RoboDK station: Conveyor Simulation.rdk

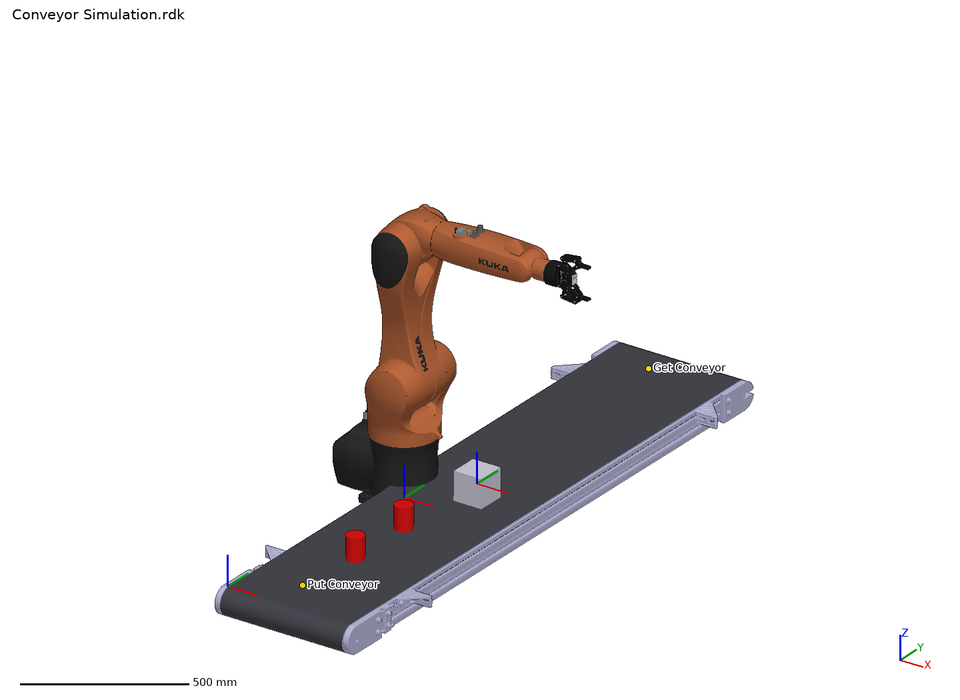
[picture v0: the station drawn from its stored meshes, robots at their saved joint values, targets as dots, program paths as lines]
Station Conveyor Simulation. Poses are relative to the parent item; angles as X-Y-Z fixed-axis rotations.
  - frame KUKA KR 10 R900 sixx Base at (-17.88, 1337.47, -86.35) mm
    - robot KUKA KR 10 R900 sixx: 6 axes, payload 10 kg, reach 901 mm, repeatability 0.03 mm, weight 52 kg
        modified DH rows (alpha deg, a mm, theta deg, d mm): 0, 0, 0, 400; -90, 25, 0, 0; 0, 455, -90, 0; -90, 35, 0, 420; 90, 0, 0, 0; -90, 0, 180, 80
        joint limits [-170, -190, -120, -185, -120, -350] to [170, 45, 156, 185, 120, 350]; home [0, -90, 90, 0, 0, 0]; saved at [0, -90, 90, 0, 0, 0]
      - tool Gripper RobotiQ 85 Opened, TCP at (0, 0, 130) mm, size 147.4 x 146.8 x 75 mm
  - frame ConveyorReference at (0, 403.83, 0) mm
    - target Get Conveyor (Cartesian target) at (200, 1882.78, 20) mm, rotated rx 90 ry 0 rz 0 deg; joints [0, 0, 0, 0, 0, 43.699]
    - target Put Conveyor (Cartesian target) at (200, 100, 20) mm, rotated rx 90 ry 0 rz -180 deg; joints [134.006, 22.86, -66.558, 43.699, -45.994, 0]
    - object Conveyor at (0, 300, -50) mm, size 597 x 2090.8 x 107.2 mm
      - Python program RunConveyor (listed below)
      - Python program WaitForPart (listed below)
      - Python program SimulateGripper (listed below)
    - object Part 1 at (200, 369.41, 40) mm, size 60 x 60 x 80 mm
    - object Part 2 at (200, 619.38, 40) mm, size 60 x 60 x 80 mm
  - frame Frame 3 at (262.28, 1312.72, 47.33) mm
    - object box at (0, 0, 0) mm, size 100 x 100 x 100 mm, geometry from box.sld

--- Python program RunConveyor ---
# Type help("robolink") or help("robodk") for more information
# Press F5 to run the script
# Note: you do not need to keep a copy of this file, your python script is saved with the station
from robolink import *    # API to communicate with RoboDK
from robodk import *      # basic matrix operations
RDK = Robolink()

# This script simulates a conveyor belt
CONVEYOR_NAME = 'Conveyor'
PICKABLE_OBJECTS_KEYWORD = 'Part'

# Speed of movement in MM/S with respect to the conveyor coordinates:
MOVE_SPEED_MMS = [0,5,0]
REFRESH_RATE = 0.005

# Define workspace of the conveyor to pick the objects:
CONV_SZ_X_MIN = 0
CONV_SZ_X_MAX = 440
CONV_SZ_Y_MIN = 0
CONV_SZ_Y_MAX = 2000
CONV_SZ_Z_MIN = -200
CONV_SZ_Z_MAX = +500

# Move objects that reached the end of the conveyor and were not picked:
FALLEN_OBJECTS = [0,0,-500]

# Get the conveyor item and reference for work space:
conv = RDK.Item(CONVEYOR_NAME)
conv_reference = conv.Parent()
poseconv = conv_reference.PoseAbs()

# One second in real life means 1 second of simulation. The simulation speed is taken from the station
SIMULATION_SPEED = 1

def is_inside_conveyor(pose):
    """Checks if a pose is inside the conveyor workspace"""
    pos = pose.Pos()
    if pos[0] > CONV_SZ_X_MIN and pos[0] < CONV_SZ_X_MAX and pos[1] > CONV_SZ_Y_MIN and pos[1] < CONV_SZ_Y_MAX and pos[2] > CONV_SZ_Z_MIN and pos[2] < CONV_SZ_Z_MAX:
        return True
    return False

def conveyor_move_object(pose, delta_time):
    """Moves the object pose through the conveyor depending on the time and speed"""
    delta_mm = mult3(MOVE_SPEED_MMS, delta_time)
    newpose = transl(delta_mm)*pose
    return newpose

# Get all objects (string list)
all_objects = RDK.ItemList(ITEM_TYPE_OBJECT, True)

# Convert object list into item pointers (faster)
# Also filter the list to take into account pickable objects only
objects = []
objects_name = []
objects_active = []
for i in range(len(all_objects)):
    if all_objects[i].count(PICKABLE_OBJECTS_KEYWORD) > 0:
        objects.append(RDK.Item(all_objects[i]))
        objects_name.append(all_objects[i])
        objects_active.append(False)

# The number of objects that can go in the conveyor
nobjects = len(objects)


# Infinite loop to simulate the conveyor behavior
current_time = 0
tic()
time_last = toc()
while True:
    # First: Look for objects that are not in the conveyor but are in the conveyor workspace
    for i in range(nobjects):
        obj_i = objects[i]

        # Skip if the object is already in the conveyor
        if objects_active[i]:
            continue

        # Check if the object has already been taken by a tool. If so, do not take it in the conveyor
        if obj_i.Parent().Type() == ITEM_TYPE_TOOL:
            continue

        # Check if the object is within the conveyor work area
        posei = obj_i.PoseAbs()
        poseirel = invH(poseconv)*posei
        if is_inside_conveyor(poseirel):
            # take the object
            obj_i.setParentStatic(conv)
            print('Adding object %s to the conveyor' % objects_name[i])
            objects_active[i] = True

    # Second step: Update the position of every object in the conveyor
    SIMULATION_SPEED = RDK.SimulationSpeed()
    time_current = toc()
    time_delta = time_current - time_last
    time_last = time_current
    current_time = current_time + time_delta*SIMULATION_SPEED

    # Make a list of objects with their matching positions to update
    obj_items = []
    obj_poses_abs = []
    for i in range(nobjects):
        obj_i = objects[i]

        # Check if the object has been picked from the conveyor
        if objects_active[i] and not obj_i.Parent().equals(conv):
            objects_active[i] = False
            print('Object %s was picked from the conveyor' % objects_name[i])
            continue

        # Skip update for objects that are not in the conveyor
        if not objects_active[i]:
            continue

        # Update the position of the object
        posei = invH(poseconv)*obj_i.PoseAbs()
        newposei = conveyor_move_object(posei, time_delta*SIMULATION_SPEED)
        if not is_inside_conveyor(newposei):
            print('Warning!! Object %s fell from the conveyor at %.1f seconds after simulation started' % (objects_name[i], current_time))
            #raise Exception('Object %s was not picked from the conveyor!' % objects_name[i])
            newposei = transl(FALLEN_OBJECTS)*newposei
            objects_active[i] = False

        #obj_i.setPose(newposei) # this will provoke a refresh (can be slow)
        obj_items.append(obj_i)
        obj_poses_abs.append(poseconv*newposei)

    # Update the object positions
    RDK.setPosesAbs(obj_items, obj_poses_abs)

    # Take a break...
    pause(REFRESH_RATE)

--- Python program WaitForPart ---
# Type help("robolink") or help("robodk") for more information
# Press F5 to run the script
# Note: you do not need to keep a copy of this file, your python script is saved with the station
from robolink import *    # API to communicate with RoboDK
from robodk import *      # basic matrix operations
RDK = Robolink()

# This script allows to simulate a laser sensor
# that detect the presence of a part in a plane,
# such as a part crossing a laser sensor in a
# conveyor belt

# The script finishes once a part has been detected
# so it works like a WAIT UNTIL function.

# Use a target from the station as a reference plane:
TARGET_NAME = 'Get Conveyor'
LASER_PLANE = [0,-1,0] # normal of the plane

# Activate within this tolerance
TOLERANCE_CHECK_MM = 10

# Look for parts with the keyword "Part"
PICKABLE_OBJECTS_KEYWORD = 'Part'

# Update status every 1 ms
RECHECK_PERIOD = 0.001

# Get the target and the detection plane
target = RDK.Item(TARGET_NAME)
targetpose = target.PoseAbs()
DETECT_PLANE_POINT = targetpose.Pos()
DETECT_PLANE_VECTOR = LASER_PLANE

# Define a function to detect a target
def part_detected(pos):
    """Check if a part is in the detection area (proximity of a point to a plane)"""
    pos_proj = proj_pt_2_plane(pos, DETECT_PLANE_POINT, DETECT_PLANE_VECTOR)
    distance2plane = norm(subs3(pos,pos_proj))
    if distance2plane < TOLERANCE_CHECK_MM:
        return True
    return False

# Get all object names
all_objects = RDK.ItemList(ITEM_TYPE_OBJECT, True)

# Get object items in a list (faster) and filter by keyword
check_objects = []
check_objects_names = []
for i in range(len(all_objects)):
    if all_objects[i].count(PICKABLE_OBJECTS_KEYWORD) > 0:
        check_objects_names.append(all_objects[i])
        check_objects.append(RDK.Item(all_objects[i]))

# Make sure that there are part that we are expecting
nCheck_objects = len(check_objects)
if nCheck_objects == 0:
    raise Exception('No parts to check for. The keyword is %s.' % PICKABLE_OBJECTS_KEYWORD)

# Loop forever until a part is detected by the sensor
part_available = False;
while not part_available:
    for i in range(nCheck_objects):
        if part_detected(check_objects[i].PoseAbs().Pos()):
            print('Part detected: %s' % check_objects_names[i])
            part_available = True
            break

    # Wait some time...
    pause(RECHECK_PERIOD)

print('Procedure finished')

--- Python program SimulateGripper ---
# Type help("robolink") or help("robodk") for more information
# Press F5 to run the script
# Note: you do not need to keep a copy of this file, your python script is saved with the station
from robolink import *    # API to communicate with RoboDK
from robodk import *      # basic matrix operations
RDK = Robolink()

# This file allows simulating the opening and closing of grippers.
# Two models of the gripper per robot are required: one opened and one closed.
# The opened model of the gripper should have the keyword "Opened"
# The closed model of the gripper should have the keyword "Closed"
# Simply place this file in the station and leave it running to
# make it work

OPENED_KEYWORD = 'Opened'
CLOSED_KEYWORD = 'Closed'
UPDATE_FREQUENCY = 0.01

# Loop forever
print('Starting infinite loop to simulate open/close of tools')
while True:
    # First step: get a list of tool pairs (open, closed) per robot
    Tool_Pairs = []
    # get all the robot names (strings)
    all_robots = RDK.ItemList(ITEM_TYPE_ROBOT)
    for i in range(len(all_robots)):
        roboti = RDK.Item(all_robots[i])
        roboti_name = roboti.Name()
        # get the tools of each robot
        roboti_tools = roboti.Childs()
        opened = None
        closed = None
        # store the opened model and closed model of each gripper
        for t in range(len(roboti_tools)):
            tnamei = roboti_tools[t].Name()
            if not isinstance(opened,Item) and tnamei.count(OPENED_KEYWORD) > 0:
                opened = roboti_tools[t]
                print('Using %s from robot %s as gripper opened' % (tnamei, roboti_name))
            elif not isinstance(closed,Item) and tnamei.count(CLOSED_KEYWORD) > 0:
                closed = roboti_tools[t]
                print('Using %s from robot %s as gripper closed' % (tnamei, roboti_name))

            if isinstance(opened, Item) and isinstance(closed, Item):
                # Stop if we have an open state and a closed state per robot
                break;
        Tool_Pairs.append([opened, closed])

    # We may find as many pairs of tools as robots are available in the station
    nTool_Pairs = len(Tool_Pairs)
    while True:
        #try:
            # Iterate through all tool pairs and detect the presence of objects
            for i in range(nTool_Pairs):
                opened = Tool_Pairs[i][0]
                closed = Tool_Pairs[i][1]
                open_valid = isinstance(opened,Item)
                close_valid = isinstance(closed,Item)
                tool_is_open = True

                # Check if the tool holds one or more objects:
                if (open_valid and len(opened.Childs()) > 0) or (close_valid and len(closed.Childs()) > 0):
                    tool_is_open = False

                # Update the visibility of the tools
                if open_valid:
                    opened.setVisible(tool_is_open)
                if close_valid:
                    closed.setVisible(not tool_is_open)

            # Take a pause...
            pause(UPDATE_FREQUENCY)

        #except:
            #print('An item was deleted. Remaking tool list')
            #break
